# B&R Automation Studio project PickupStation (part 2)

#### Actions.st
```iecst
ACTION SetInitialValuesAction:

	gHMI.AutomaticPage.StamperOffset := gStamper.Parameters.Offset;
	gHMI.AutomaticPage.ConveyorSpeed := gConveyor.Parameters.TargetSpeed;
	gHMI.AutomaticPage.StamperIncludedCheckbox := gMainMachine.Parameters.StamperEnable;
	gHMI.ManualPage.ConveyorAcceleration := gConveyor.Parameters.Acceleration;
	gHMI.ManualPage.ConveyorSpeed := gConveyor.Commands.Manual.Speed;
	gHMI.ManualPage.StamperPosition := gStamper.Commands.Manual.Position;
	gHMI.ManualPage.StamperSpeed := gStamper.Commands.Manual.Speed;
	gHMI.ManualPage.StamperAcceleration := gStamper.Parameters.Acceleration;

END_ACTION

ACTION AutomaticPageAction:

	// Link button
	IF gMainMachine.Feedbacks.WaitModeSelection
		OR gMainMachine.Feedbacks.Error
		OR gMainMachine.Feedbacks.WaitingInit
		OR gMainMachine.Feedbacks.WaitingStart
		OR gMainMachine.Feedbacks.ManualMode THEN

		gHMI.AutomaticPage.LinkButtonEnable := TRUE;
		gMainMachine.Commands.LinkMode := gHMI.AutomaticPage.LinkButton;
	ELSE
		gHMI.AutomaticPage.LinkButtonEnable := FALSE;
	END_IF

	// Init button
	IF NOT gMainMachine.Commands.LinkMode THEN

		IF gMainMachine.Commands.Automatic.Init AND gMainMachine.Feedbacks.InitDone THEN
			gHMI.AutomaticPage.InitButton := FALSE;
			gMainMachine.Commands.Automatic.Init := FALSE;
		END_IF

		IF gMainMachine.Feedbacks.WaitingInit OR gMainMachine.Feedbacks.Error THEN

			gHMI.AutomaticPage.InitButtonEnable := TRUE;
		ELSE
			gHMI.AutomaticPage.InitButtonEnable := FALSE;
			gHMI.AutomaticPage.InitButton := FALSE;
		END_IF
		gMainMachine.Commands.Automatic.Init := gHMI.AutomaticPage.InitButton;
	ELSE
		gHMI.AutomaticPage.InitButtonEnable := FALSE;
		gHMI.AutomaticPage.InitButton := FALSE;
	END_IF
	IF EDGEPOS(gMainMachine.Commands.Automatic.Init) THEN
		gHMI.AutomaticPage.AutoButton := TRUE;
	END_IF

	// AskRemoveCaps
	IF NOT gMainMachine.Commands.LinkMode THEN
		gHMI.AutomaticPage.AskRemoveCaps := gMainMachine.Feedbacks.AskRemoveCaps;
		IF gHMI.AutomaticPage.CapsRemoved THEN
			gMainMachine.Commands.Automatic.CapsRemoved := TRUE;
			gHMI.AutomaticPage.CapsRemoved := FALSE;
		END_IF
		IF NOT gMainMachine.Feedbacks.AskRemoveCaps THEN
			gMainMachine.Commands.Automatic.CapsRemoved := FALSE;
		END_IF
	ELSE
		gHMI.AutomaticPage.CapsRemoved := FALSE;
		gHMI.AutomaticPage.AskRemoveCaps := FALSE;
	END_IF

	// Auto button
	IF NOT gMainMachine.Commands.LinkMode THEN
		IF gMainMachine.Feedbacks.WaitModeSelection OR NOT gMainMachine.Feedbacks.Started THEN

			gHMI.AutomaticPage.AutoButtonEnable := TRUE;
			gMainMachine.Commands.Automatic.Enable := gHMI.AutomaticPage.AutoButton;
		ELSE
			gHMI.AutomaticPage.AutoButtonEnable := FALSE;
		END_IF
	ELSE
		gHMI.AutomaticPage.AutoButtonEnable := FALSE;
		gHMI.AutomaticPage.AutoButton := FALSE;
	END_IF
	IF EDGEPOS(gMainMachine.Commands.Automatic.Enable) THEN
		gHMI.ManualPage.ManualButton := FALSE;
	END_IF

	// Start button
	IF NOT gMainMachine.Commands.LinkMode THEN

		IF gMainMachine.Feedbacks.WaitingStart THEN

			gHMI.AutomaticPage.StartButtonEnable := TRUE;
			gHMI.AutomaticPage.StopButtonVisibility := FALSE;

		ELSIF gMainMachine.Feedbacks.Started AND gMainMachine.Commands.Automatic.Start THEN

			gHMI.AutomaticPage.StartButtonEnable := FALSE;
			gHMI.AutomaticPage.StopButtonVisibility := TRUE;
		ELSE
			gHMI.AutomaticPage.StartButtonEnable := FALSE;
			gHMI.AutomaticPage.StopButtonVisibility := FALSE;
			gHMI.AutomaticPage.StartButton := FALSE;
		END_IF

		gMainMachine.Commands.Automatic.Start := gHMI.AutomaticPage.StartButton;

	ELSE
		gHMI.AutomaticPage.StartButtonEnable := FALSE;
		gHMI.AutomaticPage.StopButtonVisibility := FALSE;
		gHMI.AutomaticPage.StartButton := FALSE;
	END_IF

	// Conveyor speed slider button
	gHMI.AutomaticPage.ConveyorSpeedEnable := NOT gMainMachine.Commands.LinkMode;
	IF NOT gMainMachine.Commands.LinkMode THEN
		gConveyor.Parameters.TargetSpeed := gHMI.AutomaticPage.ConveyorSpeed;
	ELSE
		gHMI.AutomaticPage.ConveyorSpeed := gConveyor.Parameters.TargetSpeed;
	END_IF

	// Ready to start
	gHMI.AutomaticPage.ReadyToStartVisibility := gMainMachine.Feedbacks.WaitingStart;

	// Clear statistics button
	IF NOT gMainMachine.Commands.LinkMode THEN
		IF NOT gMainMachine.Feedbacks.ClearStatsDone THEN
			gMainMachine.Commands.ClearStats := gHMI.AutomaticPage.ClearStats;
		ELSE
			gMainMachine.Commands.ClearStats := FALSE;
			gHMI.AutomaticPage.ClearStats := FALSE;
		END_IF
	END_IF

	// Statistics
	gHMI.AutomaticPage.CapsCounter := gMainMachine.Statistics.CapsCounter;
	gHMI.AutomaticPage.CurrentCapWorkingTime := TIME_TO_UDINT(gMainMachine.Statistics.CurrentCapWorkingTime);
	gHMI.AutomaticPage.LastCapWorkedTime := TIME_TO_UDINT(gMainMachine.Statistics.LastCapWorkingTime);
	gHMI.AutomaticPage.AvgCapWorkTime := TIME_TO_UDINT(gMainMachine.Statistics.AverageCapWorkingTime);

	// Stamper offset slider button
	IF NOT gMainMachine.Commands.LinkMode THEN

		gHMI.AutomaticPage.StamperOffsetEnable := TRUE;
		gStamper.Parameters.Offset := gHMI.AutomaticPage.StamperOffset;

	ELSE
		gHMI.AutomaticPage.StamperOffsetEnable := FALSE;
		gHMI.AutomaticPage.StamperOffset := gStamper.Parameters.Offset;
	END_IF

	// Stamper inclusion
	IF NOT gMainMachine.Commands.LinkMode THEN
		gHMI.AutomaticPage.StamperIncludedCheckboxEnable := TRUE;
		gMainMachine.Parameters.StamperEnable := gHMI.AutomaticPage.StamperIncludedCheckbox;
	ELSE
		gHMI.AutomaticPage.StamperIncludedCheckboxEnable := FALSE;
		gHMI.AutomaticPage.StamperIncludedCheckbox := gMainMachine.Parameters.StamperEnable;
	END_IF

END_ACTION

ACTION HeaderContentAction:

	gHMI.HeaderContent.PendingAlarms := UDINT_TO_STRING(MIN(999,gAlarms.Feedbacks.Pendings));

	gHMI.HeaderContent.MasterConnectionOk := gMainMachine.Feedbacks.LinkOk;

	gHMI.HeaderContent.StateWaitModeSelection := gMainMachine.Feedbacks.WaitModeSelection;
	gHMI.HeaderContent.StateManual := gMainMachine.Feedbacks.ManualMode;
	gHMI.HeaderContent.StateDeliveringCap := gMainMachine.Feedbacks.DeliveringCap;
	gHMI.HeaderContent.StateError := gMainMachine.Feedbacks.Error;
	gHMI.HeaderContent.StateInitializing := gMainMachine.Feedbacks.Initializing;
	gHMI.HeaderContent.StatePickingCap := gMainMachine.Feedbacks.PickingCap;
	gHMI.HeaderContent.StatePushingCap := gMainMachine.Feedbacks.PushingCap;
	gHMI.HeaderContent.StateDeliveringCap := gMainMachine.Feedbacks.DeliveringCap;
	gHMI.HeaderContent.StateWaitingModulesReady := gMainMachine.Feedbacks.WaitingModulesReady;
	gHMI.HeaderContent.StateWaitingStart := gMainMachine.Feedbacks.WaitingStart;
	gHMI.HeaderContent.StateWaitingInit := gMainMachine.Feedbacks.WaitingInit;

	IF gMainMachine.Feedbacks.Error AND NOT gMainMachine.Commands.LinkMode THEN
		IF gHMI.HeaderContent.ResetAlarms THEN
			gMainMachine.Commands.Reset := TRUE;
		END_IF
	ELSE
		gHMI.HeaderContent.ResetAlarms := FALSE;
	END_IF

	AlarmBlinkTimer(IN:=NOT AlarmBlinkTimer.Q,PT:=T#500MS);
	IF gMainMachine.Feedbacks.Error THEN
		IF AlarmBlinkTimer.Q THEN
			gHMI.HeaderContent.AlarmBlink := NOT gHMI.HeaderContent.AlarmBlink;
		END_IF
	ELSE
		gHMI.HeaderContent.AlarmBlink := FALSE;
	END_IF
END_ACTION

ACTION ManualPageAction:

	// Manual button
	IF NOT gMainMachine.Commands.LinkMode THEN
		IF gMainMachine.Feedbacks.WaitModeSelection OR NOT gMainMachine.Feedbacks.Started THEN

			gHMI.ManualPage.ManualButtonEnable := TRUE;
			gMainMachine.Commands.Manual.Enable := gHMI.ManualPage.ManualButton;
		ELSE
			gHMI.ManualPage.ManualButtonEnable := FALSE;
		END_IF
	ELSE
		gHMI.ManualPage.ManualButtonEnable := FALSE;
		gHMI.ManualPage.ManualButton := FALSE;
	END_IF
	IF EDGEPOS(gMainMachine.Commands.Manual.Enable) THEN
		gHMI.AutomaticPage.AutoButton := FALSE;
	END_IF

	// Push button
	IF NOT gMainMachine.Commands.LinkMode AND gMainMachine.Feedbacks.ManualMode THEN

		gHMI.ManualPage.PushCapButtonEnable := NOT (gPusher.Interface.Inputs.CapAtPickPosition XOR gPusher.Interface.Inputs.MagazineEmpty);
		gPusher.Commands.Manual.Push := gHMI.ManualPage.PushCapButton;

	ELSE
		gHMI.ManualPage.PushCapButtonEnable := FALSE;
		gHMI.ManualPage.PushCapButton := FALSE;
	END_IF

	// Picker forward button
	IF NOT gMainMachine.Commands.LinkMode AND gMainMachine.Feedbacks.ManualMode THEN

		gHMI.ManualPage.ArmForwardButtonEnable := NOT gPusher.Interface.Inputs.CapAtPickPosition OR (gPusher.Interface.Inputs.CapAtPickPosition AND NOT gPicker.Commands.Manual.ActivateGrip);
		gPicker.Commands.Manual.MoveForward := gHMI.ManualPage.ArmForwardButton;

	ELSE
		gHMI.ManualPage.ArmForwardButtonEnable := FALSE;
		gHMI.ManualPage.ArmForwardButton := FALSE;
	END_IF

	// Picker backward button
	IF NOT gMainMachine.Commands.LinkMode AND gMainMachine.Feedbacks.ManualMode THEN

		gHMI.ManualPage.ArmBackwardButtonEnable := NOT gHMI.ManualPage.ArmForwardButton AND NOT gConveyor.Interface.Inputs.CapInStartPosition;
		gPicker.Commands.Manual.MoveBackward := gHMI.ManualPage.ArmBackwardButton;

	ELSE
		gHMI.ManualPage.ArmBackwardButtonEnable := FALSE;
		gHMI.ManualPage.ArmBackwardButton := FALSE;
	END_IF

	// Picker vaacum button
	IF NOT gMainMachine.Commands.LinkMode AND gMainMachine.Feedbacks.ManualMode THEN

		gHMI.ManualPage.ArmVaacumButtonEnable := (gPusher.Interface.Inputs.CapAtPickPosition AND gPicker.Interface.Inputs.ArmForward) OR (gPicker.Interface.Inputs.ArmBackward AND gPicker.Commands.Manual.ActivateGrip);
		gPicker.Commands.Manual.ActivateGrip := gHMI.ManualPage.ArmVaacumButton;

	ELSE
		gHMI.ManualPage.ArmVaacumButtonEnable := FALSE;
		gHMI.ManualPage.ArmVaacumButton := FALSE;
	END_IF

	// Conveyor home button
	IF NOT gMainMachine.Commands.LinkMode AND gMainMachine.Feedbacks.ManualMode THEN

		gHMI.ManualPage.ConveyorHomeButtonEnable := TRUE;
		gConveyor.Commands.Manual.Home := gHMI.ManualPage.ConveyorHomeButton;

	ELSE
		gHMI.ManualPage.ConveyorHomeButtonEnable := FALSE;
		gHMI.ManualPage.ConveyorHomeButton := FALSE;
	END_IF
	gHMI.ManualPage.ConveyorAxisHomed := gConveyor.Feedbacks.AxisHomed;

	// Conveyor power button
	IF NOT gMainMachine.Commands.LinkMode AND gMainMachine.Feedbacks.ManualMode THEN

		gHMI.ManualPage.ConveyorPowerButtonEnable := gConveyor.Feedbacks.AxisHomed;
		gConveyor.Commands.Manual.PowerOn := gHMI.ManualPage.ConveyorPowerButton;

	ELSE
		gHMI.ManualPage.ConveyorPowerButtonEnable := FALSE;
		gHMI.ManualPage.ConveyorPowerButton := FALSE;
	END_IF
	gHMI.ManualPage.ConveyorAxisPowered := gConveyor.Feedbacks.AxisPowered;

	// Conveyor move button
	IF NOT gMainMachine.Commands.LinkMode AND gMainMachine.Feedbacks.ManualMode THEN

		gHMI.ManualPage.ConveyorMoveButtonEnable := gConveyor.Feedbacks.AxisHomed AND gConveyor.Feedbacks.AxisPowered AND (gConveyor.Commands.Manual.Speed>0 OR NOT gConveyor.Interface.Inputs.CapInStartPosition);
		gConveyor.Commands.Manual.Move := gHMI.ManualPage.ConveyorMoveButton;

	ELSE
		gHMI.ManualPage.ConveyorMoveButtonEnable := FALSE;
		gHMI.ManualPage.ConveyorMoveButton := FALSE;
	END_IF

	// Conveyor speed
	IF NOT gMainMachine.Commands.LinkMode AND gMainMachine.Feedbacks.ManualMode THEN

		gHMI.ManualPage.ConveyorSpeedEnable := NOT gConveyor.Commands.Manual.Move;
		gConveyor.Commands.Manual.Speed := gHMI.ManualPage.ConveyorSpeed;

	ELSE
		gHMI.ManualPage.ConveyorSpeedEnable := FALSE;
		gHMI.ManualPage.ConveyorSpeed := gConveyor.Commands.Manual.Speed;
	END_IF

	// Conveyor acceleration
	IF NOT gMainMachine.Commands.LinkMode AND gMainMachine.Feedbacks.ManualMode THEN

		gHMI.ManualPage.ConveyorAccelerationEnable := NOT gConveyor.Commands.Manual.Move;
		gConveyor.Parameters.Acceleration := gHMI.ManualPage.ConveyorAcceleration;
	ELSE
		gHMI.ManualPage.ConveyorAccelerationEnable := FALSE;
		gHMI.ManualPage.ConveyorAcceleration := gConveyor.Parameters.Acceleration;
	END_IF

	// Stamper home button
	IF NOT gMainMachine.Commands.LinkMode AND gMainMachine.Feedbacks.ManualMode THEN

		gHMI.ManualPage.StamperHomeButtonEnable := TRUE;
		gStamper.Commands.Manual.Home := gHMI.ManualPage.StamperHomeButton;

	ELSE
		gHMI.ManualPage.StamperHomeButtonEnable := FALSE;
		gHMI.ManualPage.StamperHomeButton := FALSE;
	END_IF
	gHMI.ManualPage.StamperAxisHomed := gStamper.Feedbacks.AxisHomed;

	// Stamper power button
	IF NOT gMainMachine.Commands.LinkMode AND gMainMachine.Feedbacks.ManualMode THEN

		gHMI.ManualPage.StamperPowerButtonEnable := gStamper.Feedbacks.AxisHomed;
		gStamper.Commands.Manual.PowerOn := gHMI.ManualPage.StamperPowerButton;

	ELSE
		gHMI.ManualPage.StamperPowerButtonEnable := FALSE;
		gHMI.ManualPage.StamperPowerButton := FALSE;
	END_IF
	gHMI.ManualPage.StamperAxisPowered := gStamper.Feedbacks.AxisPowered;

	// Stamper move button
	IF NOT gMainMachine.Commands.LinkMode AND gMainMachine.Feedbacks.ManualMode THEN

		gHMI.ManualPage.StamperMoveButtonEnable := gStamper.Feedbacks.AxisHomed AND gStamper.Feedbacks.AxisPowered;
		gStamper.Commands.Manual.Move := gHMI.ManualPage.StamperMoveButton;

	ELSE
		gHMI.ManualPage.StamperMoveButtonEnable := FALSE;
		gHMI.ManualPage.StamperMoveButton := FALSE;
	END_IF

	// Stamper speed
	IF NOT gMainMachine.Commands.LinkMode AND gMainMachine.Feedbacks.ManualMode THEN

		gHMI.ManualPage.StamperSpeedEnable := NOT gStamper.Commands.Manual.Move;
		gStamper.Commands.Manual.Speed := gHMI.ManualPage.StamperSpeed;

	ELSE
		gHMI.ManualPage.StamperSpeedEnable := FALSE;
		gHMI.ManualPage.StamperSpeed := gStamper.Commands.Manual.Speed;
	END_IF

	// Stamper acceleration
	IF NOT gMainMachine.Commands.LinkMode AND gMainMachine.Feedbacks.ManualMode THEN

		gHMI.ManualPage.StamperAccelerationEnable := NOT gConveyor.Commands.Manual.Move;
		gStamper.Parameters.Acceleration := gHMI.ManualPage.StamperAcceleration;
	ELSE
		gHMI.ManualPage.StamperAccelerationEnable := FALSE;
		gHMI.ManualPage.StamperAcceleration := gStamper.Parameters.Acceleration;
	END_IF

	// Stamper position slider button
	IF NOT gMainMachine.Commands.LinkMode AND gMainMachine.Feedbacks.ManualMode THEN

		gHMI.ManualPage.StamperPositionEnable := NOT gStamper.Commands.Manual.Move;
		gStamper.Commands.Manual.Position := gHMI.ManualPage.StamperPosition;

	ELSE
		gHMI.ManualPage.StamperPositionEnable := FALSE;
		gHMI.ManualPage.StamperPosition := gStamper.Commands.Manual.Position;
	END_IF

	// Sensors
	gHMI.ManualPage.PusherInterface := gPusher.Interface;
	gHMI.ManualPage.PickerInterface := gPicker.Interface;
	gHMI.ManualPage.ConveyorInterface := gConveyor.Interface;
	gHMI.ManualPage.StamperInterface := gStamper.Interface;

	// Motion Feedback
	gHMI.ManualPage.ConveyorActPosition := gConveyor.Feedbacks.AxisPosition;
	gHMI.ManualPage.ConveyorActSpeed := gConveyor.Feedbacks.AxisSpeed;

	gHMI.ManualPage.StamperActPosition := gStamper.Feedbacks.AxisPosition;
	gHMI.ManualPage.StamperActSpeed := gStamper.Feedbacks.AxisSpeed;

END_ACTION
```

### MasterGlobalTypes.typ
```iecst
TYPE
	MasterType : 	STRUCT  (*Master Main type*)
		Inputs : MasterInputsType;
		Outputs : MasterOutputsType;
	END_STRUCT;
	MasterInputsType : 	STRUCT  (*Master Commands type*)
		HeartBeat : BOOL;
		Error : BOOL;
		WaitingStart : BOOL;
		WaitingModeSelection : BOOL;
		WaitingInit : BOOL;
		InitDone : BOOL;
		Started : BOOL;
		ClearStatsDone : BOOL;
		LinkActive : BOOL;
		ActStampIncluded : BOOL;
		ActStampOffset : REAL;
		CapsOnConveyor : USINT;
	END_STRUCT;
	MasterOutputsType : 	STRUCT  (*Master Feedbacks type*)
		HeartBeat : BOOL;
		Reset : BOOL;
		Error : BOOL;
		ClearStats : BOOL;
		Init : BOOL;
		Start : BOOL;
		AutomaticMode : BOOL;
		StampIncluded : BOOL;
		StampOffset : REAL;
		ConveyorSpeed : REAL;
	END_STRUCT;
END_TYPE
```

### MasterGlobalVariables.var
```iecst
VAR
    gMaster : MasterType;
END_VAR
```

### Program Logical/Source/Master/MasterProgram (IEC)

#### Main.st - Init, cyclic, exit code
```iecst
//******************************************************************************************************
// Program: 	HMIProgram
// Author: 		Andrea Pennisi
// Rev.: 		1.0.0
// Date:		5.12.2023
//
// Description:
// This module is used to manage the interface between Master and MainMachine
// Interface comunication protocol is OPCUA. This station is the client.
//******************************************************************************************************
PROGRAM _INIT

END_PROGRAM

PROGRAM _CYCLIC

	// MainMachine -> Master
	gMaster.Inputs.ClearStatsDone := gMainMachine.Feedbacks.ClearStatsDone;
	gMaster.Inputs.Error := gMainMachine.Feedbacks.Error;
	gMaster.Inputs.InitDone := gMainMachine.Feedbacks.InitDone;
	gMaster.Inputs.Started := gMainMachine.Feedbacks.Started;
	gMaster.Inputs.WaitingStart := gMainMachine.Feedbacks.WaitingStart;
	gMaster.Inputs.WaitingInit := gMainMachine.Feedbacks.WaitingInit;
	gMaster.Inputs.WaitingModeSelection := gMainMachine.Feedbacks.WaitModeSelection;
	gMaster.Inputs.HeartBeat := gMainMachine.Feedbacks.HeartBeat;
	gMaster.Inputs.ActStampIncluded := gMainMachine.Parameters.StamperEnable;
	gMaster.Inputs.ActStampOffset := gStamper.Parameters.Offset;
	gMaster.Inputs.LinkActive := gMainMachine.Commands.LinkMode;
	gMaster.Inputs.CapsOnConveyor := gMainMachine.Feedbacks.CapsOnConveyor;

	gMainMachine.Commands.HeartBeat := gMaster.Outputs.HeartBeat;

	IF NOT gMainMachine.Commands.LinkMode THEN
		RETURN;
	END_IF

	// Master -> MainMachine
	gMainMachine.Commands.Reset := gMaster.Outputs.Reset;
	gMainMachine.Commands.ClearStats := gMaster.Outputs.ClearStats;

	gMainMachine.Commands.Automatic.Enable := gMaster.Outputs.AutomaticMode;
	IF gMaster.Outputs.AutomaticMode THEN
		gMainMachine.Commands.Manual.Enable := FALSE;
	END_IF
	gMainMachine.Commands.Automatic.Init := gMaster.Outputs.Init;
	gMainMachine.Commands.Automatic.Start := gMaster.Outputs.Start;

	gConveyor.Parameters.TargetSpeed := gMaster.Outputs.ConveyorSpeed;
	gMainMachine.Parameters.StamperEnable := gMaster.Outputs.StampIncluded;
	gStamper.Parameters.Offset := gMaster.Outputs.StampOffset;

	IF gMaster.Outputs.Error AND NOT gMainMachine.Feedbacks.Error AND NOT gMainMachine.Commands.Reset THEN
		MpAlarmXSet(gAlarmXCoreMpLink,'MasterInError');
	END_IF

END_PROGRAM

PROGRAM _EXIT

END_PROGRAM
```

- Visualisation Logical/mappView (not shown)

- Project.language (not shown)
